% RSLogix 500 project PROC1_MATH.RSS, saved by version 8.30.00.16 %
PROJECT "PROC1"    % processor: Bul.1763 MicroLogix 1100 Series B %

PROGRAM FILES
  LAD 2 "MAIN"  3 rungs
  LAD 3 "MATH OPS"  9 rungs  % Math instructions %
  LAD 4 "VARIABLES"  9 rungs  % Stores assigned variables %

DATA FILES
  O0 OUTPUT  4 elements
  I1 INPUT  6 elements
  S2 STATUS  66 elements
  B3 BINARY  1 elements
  T4 TIMER  1 elements
  C5 COUNTER  1 elements
  R6 CONTROL  1 elements
  N7 INTEGER  28 elements
  F8 FLOAT  1 elements

LADDER 2 "MAIN"
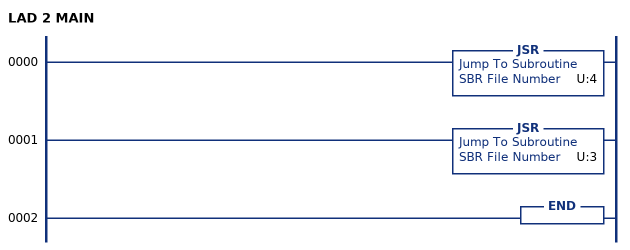
% Rung: 0 %
SOR JSR U:4 EOR
% Rung: 1 %
SOR JSR U:3 EOR
% Rung: 2 %
SOR END EOR

LADDER 3 "MATH OPS"    % Math instructions %
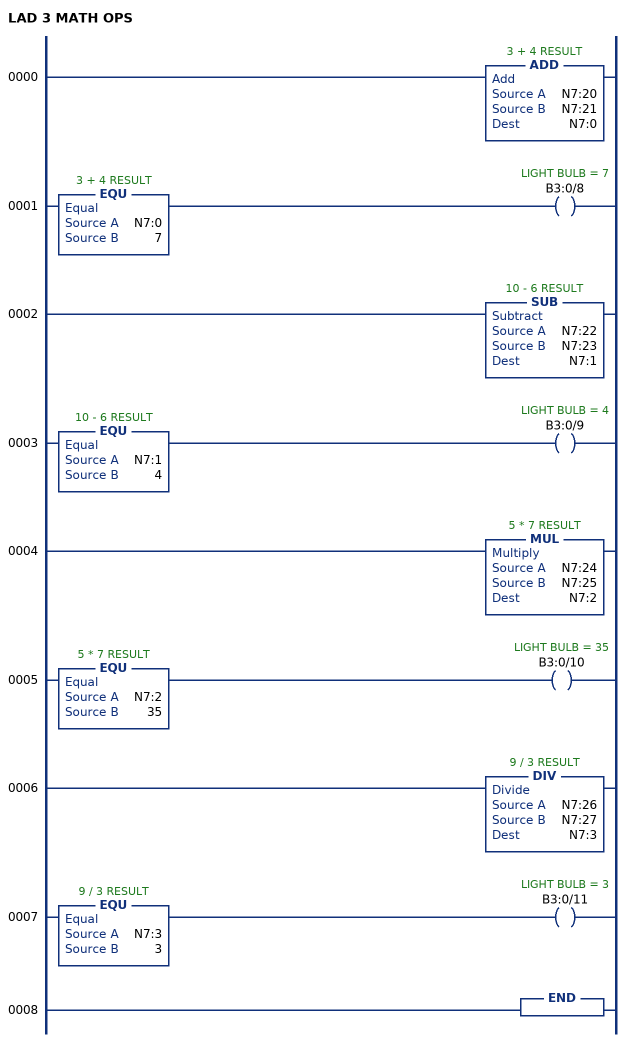
% Rung: 0 %
SOR ADD N7:20 N7:21 N7:0 EOR
%   N7:20  "Assign 3 to N7:20" %
%   N7:21  "Assign 4 to N7:21" %
%   N7:0  "3 + 4 RESULT" %
% Rung: 1 %
SOR EQU N7:0 7 OTE B3:0/8 EOR
%   N7:0  "3 + 4 RESULT" %
%   B3:0/8  "LIGHT BULB = 7" %
% Rung: 2 %
SOR SUB N7:22 N7:23 N7:1 EOR
%   N7:22  "Assign 10 to N7:22" %
%   N7:23  "Assign 6 to N7:23" %
%   N7:1  "10 - 6 RESULT" %
% Rung: 3 %
SOR EQU N7:1 4 OTE B3:0/9 EOR
%   N7:1  "10 - 6 RESULT" %
%   B3:0/9  "LIGHT BULB = 4" %
% Rung: 4 %
SOR MUL N7:24 N7:25 N7:2 EOR
%   N7:24  "Assign 5 to N7:25" %
%   N7:25  "Assign 7 to N7:25" %
%   N7:2  "5 * 7 RESULT" %
% Rung: 5 %
SOR EQU N7:2 35 OTE B3:0/10 EOR
%   N7:2  "5 * 7 RESULT" %
%   B3:0/10  "LIGHT BULB = 35" %
% Rung: 6 %
SOR DIV N7:26 N7:27 N7:3 EOR
%   N7:26  "Assign 9 to N7:26" %
%   N7:27  "Assign 3 to N7:27" %
%   N7:3  "9 / 3 RESULT" %
% Rung: 7 %
SOR EQU N7:3 3 OTE B3:0/11 EOR
%   N7:3  "9 / 3 RESULT" %
%   B3:0/11  "LIGHT BULB = 3" %
% Rung: 8 %
SOR END EOR

LADDER 4 "VARIABLES"    % Stores assigned variables %
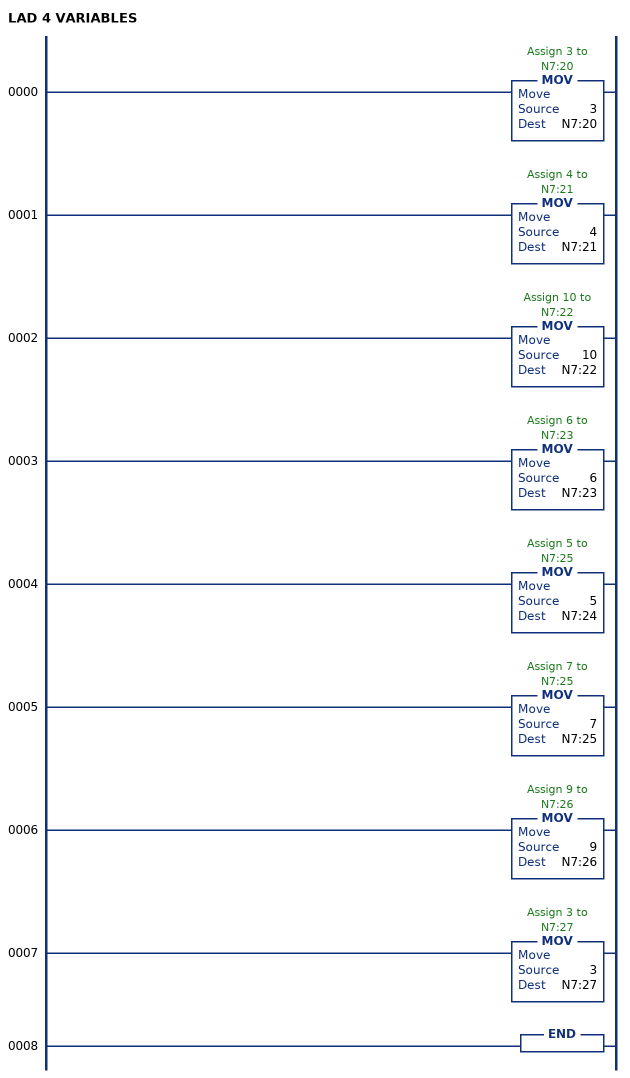
% Rung: 0 %
SOR MOV 3 N7:20 EOR
%   N7:20  "Assign 3 to N7:20" %
% Rung: 1 %
SOR MOV 4 N7:21 EOR
%   N7:21  "Assign 4 to N7:21" %
% Rung: 2 %
SOR MOV 10 N7:22 EOR
%   N7:22  "Assign 10 to N7:22" %
% Rung: 3 %
SOR MOV 6 N7:23 EOR
%   N7:23  "Assign 6 to N7:23" %
% Rung: 4 %
SOR MOV 5 N7:24 EOR
%   N7:24  "Assign 5 to N7:25" %
% Rung: 5 %
SOR MOV 7 N7:25 EOR
%   N7:25  "Assign 7 to N7:25" %
% Rung: 6 %
SOR MOV 9 N7:26 EOR
%   N7:26  "Assign 9 to N7:26" %
% Rung: 7 %
SOR MOV 3 N7:27 EOR
%   N7:27  "Assign 3 to N7:27" %
% Rung: 8 %
SOR END EOR

OTHER DOCUMENTED ADDRESSES
  B3:0/0  "TRIGGER"

REVISION NOTES
  0: Initial code
  1: Added branches
  2: More code
  3: Moved MOV commands to VARIABLES ladder
  4: Added JSR to LAD-4
